# EPICS substitutions: apps/mmfeuApp/Db/mmfeucrateFTT.substitutions
#
file "db/mmfeucrate.db" {
        pattern { P, C, PORT}
                {"B_DET_FTT_FEU", "1", "L1"  }
                {"B_DET_FTT_FEU", "2", "L1"  }
                {"B_DET_FTT_FEU", "3", "L1"  }
}
